PROGRAM prgPV
VAR
	fbPVvirt	: FB_Light;
	bPVOn		: BOOL; //{#lynus.ag#()}
	bPVOff		: BOOL; //{#lynus.ag#()}
	bStatePV	: BOOL; //{#lynus.ag#()}
	lrPVpower	: LREAL; //{#lynus.ag#()}
END_VAR

fbPVvirt(bOn:=bPVOn, bOff:=bPVOff, bLight=>bStatePV);

IF bStatePV THEN
	lrPVpower := 9.72;
	ELSE
	lrPVpower := 0;
END_IF

END_PROGRAM

(* stored: Version 1.1.0.1, ProductVersion 3.1.4024.9
   POU prgPV: Id {20f66be7-e12d-4934-98ef-69d1fde46027}, SpecialFunc None *)
